FUNCTION_BLOCK PUBLIC FB_Controller
VAR
	fbActualValue		: FB_AnalogValue;
	_refActiveLamp		: REFERENCE TO FB_Lamp;
END_VAR

IF (__ISVALIDREF(_refActiveLamp)) THEN
	_refActiveLamp();
END_IF

// Reduces the control value by 5 in the range of 10 to 100.
METHOD PUBLIC DimDown
IF (__ISVALIDREF(_refActiveLamp)) THEN
	_refActiveLamp.DimDown();
END_IF
END_METHOD

// Increments the control value by 5 in the range of 10 to 100.
METHOD PUBLIC DimUp
IF (__ISVALIDREF(_refActiveLamp)) THEN
	_refActiveLamp.DimUp();
END_IF
END_METHOD

{attribute 'monitoring' := 'call'}
PROPERTY PUBLIC nOperatingTime : DINT
GET
IF (__ISVALIDREF(_refActiveLamp)) THEN	
	nOperatingTime := _refActiveLamp.nOperatingTime;
END_IF
END_GET
SET
IF (__ISVALIDREF(_refActiveLamp)) THEN
	_refActiveLamp.nOperatingTime := nOperatingTime;
END_IF
END_SET
END_PROPERTY

// Sets the control value to 0.
METHOD PUBLIC Off
IF (__ISVALIDREF(_refActiveLamp)) THEN
	_refActiveLamp.Off();
END_IF
END_METHOD

// Sets the control value to 100.
METHOD PUBLIC On
IF (__ISVALIDREF(_refActiveLamp)) THEN
	_refActiveLamp.On();
END_IF
END_METHOD

{attribute 'monitoring' := 'call'}
PROPERTY PUBLIC refActiveLamp : REFERENCE TO FB_Lamp
GET
refActiveLamp REF= _refActiveLamp;
END_GET
SET
IF (__ISVALIDREF(_refActiveLamp)) THEN
	_refActiveLamp.Detach();
END_IF

_refActiveLamp REF= refActiveLamp;

IF (__ISVALIDREF(refActiveLamp)) THEN
	refActiveLamp.Attach(fbActualValue);
END_IF
END_SET
END_PROPERTY

END_FUNCTION_BLOCK

(* stored: Version 1.1.0.1, ProductVersion 3.1.4024.11
   POU FB_Controller: Id {057b5bd1-e33b-44a4-8eb0-93b60ce9e81d}, SpecialFunc None
   Method DimDown: Id {130de151-930d-42fb-84c7-94f9e80ef2d1}
   Method DimUp: Id {6fad7f57-9367-4e6e-ba7a-7dfd0e3aeed8}
   Property nOperatingTime: Id {ab119408-4e98-4501-8fc6-262fd96347a7}
   Get Get: Id {9952d302-4260-408a-93bc-b9e54131b4da}
   Set Set: Id {5a9b9b01-5d71-48fa-bfa1-5ddab2a9368b}
   Method Off: Id {9d5e0538-50dd-4f19-a271-b30075978c0e}
   Method On: Id {89c7d278-6585-48c0-967a-839fca58784f}
   Property refActiveLamp: Id {ec0f52a6-c70f-42f8-9c3a-71f12596d6fa}
   Get Get: Id {a21c5761-4c53-497c-bcc5-11c88e64a910}
   Set Set: Id {a6e8f2a1-2c1c-402e-abad-b72a09e11163} *)
